TYPE Sfts_Inputs_DUT :
STRUCT
	DP_Extended:  BOOL;
	DP_Retracted:  Bool;
END_STRUCT
END_TYPE

(* stored: Version 1.1.0.1
   DUT Sfts_Inputs_DUT: Id {ba2ebe3e-c23d-41a9-8f87-fd42b7489f40} *)
